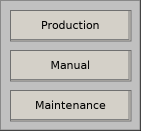
VISUALIZATION VFM_OperatingMode  // 141x131
VAR_IN_OUT
	HMI : ST_PackMLBaseModule_HMI;
END_VAR
    Rectangle (0,0 141x131)
    Button (10,10 121x31), "Production", colour toggle: HMI.Status.Mode = E_PMLUnitMode.ePMLUnitMode_Production
        OnMouseClick: execute { HMI.Command.Mode := E_PMLUnitMode.ePMLUnitMode_Production; }
    Button (10,50 121x31), "Manual", colour toggle: HMI.Status.Mode = E_PMLUnitMode.ePMLUnitMode_Manual
        OnMouseClick: execute { HMI.Command.Mode := E_PMLUnitMode.ePMLUnitMode_Manual; }
    Button (10,90 121x31), "Maintenance", colour toggle: HMI.Status.Mode = E_PMLUnitMode.ePMLUnitMode_Maintenance
        OnMouseClick: execute { HMI.Command.Mode := E_PMLUnitMode.ePMLUnitMode_Maintenance; }
END_VISUALIZATION

(* stored: Version 1.1.0.1, ProductVersion 3.1.4024.12
   Visu VFM_OperatingMode: Id {5d7b1ce3-02f7-499d-94d2-86f82ac8c510} *)
